PROGRAM Main
VAR
	fbWriteWstrToFile_0	:BFB_WriteWstrToFile;
	fbWriteStrToFile_0	:BFB_WriteStrToFile;
	
	sStr				:STRING := 'D:\BeckhoffBox\TestNotepad.txt';
	sStr1				:STRING := 'D:\BeckhoffBox\TestStrNotepad.txt';
	aWstr				:ARRAY[0..19] OF WSTRING := ["第一行", 18("中间行"), "最后一行"];
	aStr				:ARRAY[0..19] OF STRING := ['First', 18('For Test'), 'Last'];
	bWrite				:BOOL;
	bWrite1				:BOOL;
	bAppend				:BOOL;
	bOpen				:BOOL;
	bClose				:BOOL;
	bSave				:BOOL;
END_VAR

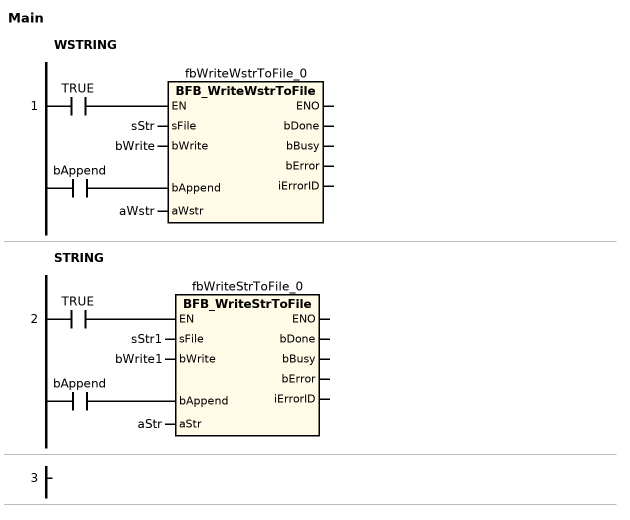
// NETWORK 1: WSTRING
fbWriteWstrToFile_0(sFile := sStr, bWrite := bWrite, bAppend := bAppend, aWstr := aWstr); // BFB_WriteWstrToFile

// NETWORK 2: STRING
fbWriteStrToFile_0(sFile := sStr1, bWrite := bWrite1, bAppend := bAppend, aStr := aStr); // BFB_WriteStrToFile

// NETWORK 3

END_PROGRAM

(* stored: Version 1.1.0.1, ProductVersion 3.1.4024.9
   POU Main: Id {24f2b17b-6006-4185-a885-aa36c4af78ad}, SpecialFunc None *)
